// TwinCAT 3 PLC project AIR_Kinematics
// ProgramVersion: 3.1.4023.0
// libraries:
//   Standard, * (System)
//   Tc2_MC2, * (Beckhoff Automation GmbH)
//   Tc2_Standard, * (Beckhoff Automation GmbH)
//   Tc2_System, * (Beckhoff Automation GmbH)
//   Tc2_Utilities, * (Beckhoff Automation GmbH)
//   Tc3_Module, * (Beckhoff Automation GmbH)
// project tree:
//   DUTs/ ST_Trajectory.TcDUT
//   GVLs/ GVL.TcGVL
//   / PlcTask.TcTTO
//   POUs/ MAIN.TcPOU
//   StateData/ MoveState_t.TcDUT
// real-time tasks:
//   TASK PlcTask: cycle T#1ms, priority 1, ADS port 350
// motion (NC):
//   TASK NC-Task 1 SAF: cycle T#1ms, priority 4, ADS port 501
//   TASK NC-Task 1 SVB: cycle T#5ms, priority 8, ADS port 511
//   AXIS Axis 1 (id 1)
//     General: UnitName=Degree
//     Dynamic: AccelerationMaximum=1500, DecelerationMaximum=1500, Acceleration=2050.2, Deceleration=2050.2, Jerk=61506
//     Velo: RefSearch=2, RefSync=2, SlowManual=10, FastManual=50, Fast=136.68, Maximum=136.68
//     PositionAreaControl: Enable=false
//     TargetPosControl: Enable=false
//     OtherSettings: AllowMotionCmdToSlave=true
//     encoder EncType=19
//       EncPara: ScaleFactorNumerator=3.6, ScaleFactorDenominator=1048576, Offset=234, MaxCount=#xffffffff, ReferenceSystem=1
//         SoftEndMinControl: Enable=true, Range=-45
//         SoftEndMaxControl: Enable=true, Range=45
//     drive DrvType=16
//       DrvPara: MaxCount=#xffffffff, DriveControlDWord=#x00020000
//         Analog: VeloReferenz=150.348, VeloScale=32, TorqueSetpointScale=10, ScaleFactorActTorque=0.1
//         TimeComp: TaskDelayCycles=1
//     controller CtrType=1
//       CtrPara: PriorControlFactor=1
//         PosDiffControl: Enable=false
//         Observer: BandWidth=20
//   AXIS Axis 2 (id 2)
//     General: UnitName=Degree
//     Dynamic: AccelerationMaximum=1500, DecelerationMaximum=1500, Acceleration=2050.2, Deceleration=2050.2, Jerk=61506
//     Velo: RefSearch=2, RefSync=2, SlowManual=5, FastManual=50, Fast=136.68, Maximum=136.68
//     PositionAreaControl: Enable=false
//     TargetPosControl: Enable=false
//     OtherSettings: AllowMotionCmdToSlave=true
//     encoder EncType=19
//       EncPara: ScaleFactorNumerator=3.6, ScaleFactorDenominator=1048576, Offset=356.451663208008, Inverse=true, MaxCount=#xffffffff, ReferenceSystem=1
//         SoftEndMinControl: Enable=true, Range=-1
//         SoftEndMaxControl: Enable=true, Range=90
//     drive DrvType=16
//       DrvPara: Inverse=true, MaxCount=#xffffffff, DriveControlDWord=#x00020000
//         Analog: VeloReferenz=150.348, VeloScale=32, TorqueSetpointScale=10, ScaleFactorActTorque=0.1
//         TimeComp: TaskDelayCycles=1
//     controller CtrType=1
//       CtrPara: PriorControlFactor=1
//         PosDiffControl: Enable=false
//         Observer: BandWidth=20
//   AXIS Axis 3 (id 3)
//     General: UnitName=Degree
//     Dynamic: AccelerationMaximum=3000, DecelerationMaximum=3000, Acceleration=4369.5, Deceleration=4369.5, Jerk=131085
//     Velo: RefSearch=2, RefSync=2, SlowManual=20, FastManual=50, Fast=291.3, Maximum=291.3
//     PositionAreaControl: Enable=false
//     TargetPosControl: Enable=false
//     OtherSettings: AllowMotionCmdToSlave=true
//     encoder EncType=19
//       EncPara: ScaleFactorNumerator=3.6, ScaleFactorDenominator=1048576, Offset=-169.531800842285, MaxCount=#xffffffff, ReferenceSystem=1
//         SoftEndMinControl: Enable=true, Range=-90
//         SoftEndMaxControl: Enable=true, Range=90
//     drive DrvType=16
//       DrvPara: MaxCount=#xffffffff, DriveControlDWord=#x00020000
//         Analog: VeloReferenz=320.43, VeloScale=32, TorqueSetpointScale=10, ScaleFactorActTorque=0.1
//         TimeComp: TaskDelayCycles=1
//     controller CtrType=1
//       CtrPara: PriorControlFactor=1
//         PosDiffControl: Enable=false
//         Observer: BandWidth=20
//   AXIS elbow (id 4)
//     Dynamic: AccelerationMaximum=300, DecelerationMaximum=300, Acceleration=1793.71, Deceleration=1793.71, Jerk=271037
//     Velo: RefSearch=2, RefSync=2, SlowManual=5, FastManual=10, Maximum=100
//     PositionAreaControl: Enable=false
//     TargetPosControl: Enable=false
//     OtherSettings: AllowMotionCmdToSlave=true
//     encoder EncType=19
//       EncPara: ScaleFactorNumerator=19.073486328125, ScaleFactorDenominator=1000000, Offset=-205.2, MaxCount=#xffffffff, ReferenceSystem=1
//         SoftEndMinControl: Enable=true, Range=12.5
//         SoftEndMaxControl: Enable=true, Range=75
//     drive DrvType=16
//       DrvPara: MaxCount=#xffffffff
//         Analog: VeloReferenz=100, TorqueSetpointScale=10, ScaleFactorActTorque=0.1
//         TimeComp: TaskDelayCycles=1
//     controller CtrType=1
//       CtrPara: PriorControlFactor=1
//         PosDiffControl: Enable=false
//         Observer: BandWidth=20
//   AXIS roll (id 7)
//     Dynamic: AccelerationMaximum=30, DecelerationMaximum=30, Acceleration=75.75, Deceleration=75.75, Jerk=76507.5
//     Velo: RefSearch=1.5, RefSync=1.5, SlowManual=3.5, FastManual=7.5, Maximum=7.5
//     OtherSettings: AllowMotionCmdToSlave=true
//     encoder EncType=19
//       EncPara: ScaleFactorNumerator=2.846789, ScaleFactorDenominator=1000000, Offset=-11.48, MaxCount=#xffffffff, ReferenceSystem=1
//         SoftEndMinControl: Enable=true, Range=-15
//         SoftEndMaxControl: Enable=true, Range=15
//     drive DrvType=16
//       DrvPara: MaxCount=#xffffffff
//         Analog: VeloReferenz=7.5, TorqueSetpointScale=10, ScaleFactorActTorque=0.1
//         TimeComp: TaskDelayCycles=1
//     controller CtrType=1
//       CtrPara: PriorControlFactor=1
//         Observer: BandWidth=20
//   AXIS pitch (id 6)
//     Dynamic: AccelerationMaximum=30, DecelerationMaximum=30, Acceleration=75.75, Deceleration=75.75, Jerk=76507.5
//     Velo: RefSearch=1.5, RefSync=1.5, SlowManual=3.5, FastManual=7.5, Maximum=7.5
//     OtherSettings: AllowMotionCmdToSlave=true
//     encoder EncType=19
//       EncPara: ScaleFactorNumerator=2.846789, ScaleFactorDenominator=1000000, Offset=35, MaxCount=#xffffffff, ReferenceSystem=1
//         SoftEndMinControl: Enable=true, Range=-30
//         SoftEndMaxControl: Enable=true, Range=15
//     drive DrvType=16
//       DrvPara: MaxCount=#xffffffff
//         Analog: VeloReferenz=7.5, TorqueSetpointScale=10, ScaleFactorActTorque=0.1
//         TimeComp: TaskDelayCycles=1
//     controller CtrType=1
//       CtrPara: PriorControlFactor=1
//         Observer: BandWidth=20
//   AXIS yaw (id 5)
//     General: UnitName=Degree
//     Dynamic: AccelerationMaximum=5500, DecelerationMaximum=5500, Acceleration=2300, Deceleration=2300, Jerk=529000
//     Velo: Maximum=220
//     PositionAreaControl: Enable=false
//     OtherSettings: AllowMotionCmdToSlave=true
//     encoder EncType=19
//       EncPara: ScaleFactorNumerator=556.2698, ScaleFactorDenominator=1000000, MaxCount=#xffffffff
//         SoftEndMaxControl: Range=180
//     drive DrvType=16
//       DrvPara: MaxCount=#xffffffff
//         Analog: VeloReferenz=220, TorqueSetpointScale=10, ScaleFactorActTorque=0.1
//         TimeComp: TaskDelayCycles=1
//     controller CtrType=1
//       CtrPara: PriorControlFactor=1
//         PosDiffControl: Enable=false
//         Observer: BandWidth=20
// I/O:
//   DEVICE Device 5 (EtherCAT), AmsNetId 192.168.225.1.6.1
//     Term 12 (EK1100) [EK1100 EtherCAT Coupler (2A E-Bus)]
//       Term 13 (EL7211-0010) [EL7211-0010 1Ch. MDP742 Servo motor output stage with OCT (50V, 4.5A RMS)]
//       Term 14 (EL7211-0010) [EL7211-0010 1Ch. MDP742 Servo motor output stage with OCT (50V, 4.5A RMS)]
//       Term 15 (EL7211-0010) [EL7211-0010 1Ch. MDP742 Servo motor output stage with OCT (50V, 4.5A RMS)]
//       Term 16 (EL7211-0010) [EL7211-0010 1Ch. MDP742 Servo motor output stage with OCT (50V, 4.5A RMS)]
//       Term 17 (EL1008) [EL1008 8Ch. Dig. Input 24V, 3ms]
//       Term 18 (EL2008) [EL2008 8Ch. Dig. Output 24V, 0.5A]
//       Term 23 (EL9011) [EL9011 End Terminal]
//     Drive 19 (Capitan Drv) [Capitan Drv]
//     Drive 20 (Capitan Drv) [Capitan Drv]
//     Drive 21 (Capitan Drv) [Capitan Drv]
//     Drive 22 (Capitan Drv) [Capitan Drv]
// variable links:
//   NC-Task 1 SAF/Axes/Axis 1 <-> Device 5 (EtherCAT)/Term 12 (EK1100)/Term 13 (EL7211-0010)
//     Drive/Inputs/In/nDcOutputTime <-> InfoData/DcOutputShift
//     Drive/Inputs/In/nState1 <-> DRV Statusword/Statusword
//     Drive/Inputs/In/nState2 <-> DRV Statusword/Statusword @bit 8
//     Drive/Inputs/In/nState4 @bit 1 <-> WcState/InputToggle
//     Drive/Inputs/In/nState4 <-> WcState/WcState
//     Drive/Outputs/Out/nCtrl1 <-> DRV Controlword/Controlword
//     Drive/Outputs/Out/nCtrl2 <-> DRV Controlword/Controlword @bit 8
//     Drive/Outputs/Out/nDataOut2 <-> DRV Target velocity/Target velocity
//     Enc/Inputs/In/nDataIn1 <-> FB Position/Position
//     Enc/Inputs/In/nDcInputTime <-> InfoData/DcInputShift
//     Enc/Inputs/In/nState4 @bit 1 <-> WcState/InputToggle
//     Enc/Inputs/In/nState4 <-> WcState/WcState
//   NC-Task 1 SAF/Axes/Axis 2 <-> Device 5 (EtherCAT)/Term 12 (EK1100)/Term 14 (EL7211-0010)
//     Drive/Inputs/In/nDcOutputTime <-> InfoData/DcOutputShift
//     Drive/Inputs/In/nState1 <-> DRV Statusword/Statusword
//     Drive/Inputs/In/nState2 <-> DRV Statusword/Statusword @bit 8
//     Drive/Inputs/In/nState4 @bit 1 <-> WcState/InputToggle
//     Drive/Inputs/In/nState4 <-> WcState/WcState
//     Drive/Outputs/Out/nCtrl1 <-> DRV Controlword/Controlword
//     Drive/Outputs/Out/nCtrl2 <-> DRV Controlword/Controlword @bit 8
//     Drive/Outputs/Out/nDataOut2 <-> DRV Target velocity/Target velocity
//     Enc/Inputs/In/nDataIn1 <-> FB Position/Position
//     Enc/Inputs/In/nDcInputTime <-> InfoData/DcInputShift
//     Enc/Inputs/In/nState4 @bit 1 <-> WcState/InputToggle
//     Enc/Inputs/In/nState4 <-> WcState/WcState
//   NC-Task 1 SAF/Axes/Axis 3 <-> Device 5 (EtherCAT)/Term 12 (EK1100)/Term 16 (EL7211-0010)
//     Drive/Inputs/In/nDcOutputTime <-> InfoData/DcOutputShift
//     Drive/Inputs/In/nState1 <-> DRV Statusword/Statusword
//     Drive/Inputs/In/nState2 <-> DRV Statusword/Statusword @bit 8
//     Drive/Inputs/In/nState4 @bit 1 <-> WcState/InputToggle
//     Drive/Inputs/In/nState4 <-> WcState/WcState
//     Drive/Outputs/Out/nCtrl1 <-> DRV Controlword/Controlword
//     Drive/Outputs/Out/nCtrl2 <-> DRV Controlword/Controlword @bit 8
//     Drive/Outputs/Out/nDataOut2 <-> DRV Target velocity/Target velocity
//     Enc/Inputs/In/nDataIn1 <-> FB Position/Position
//     Enc/Inputs/In/nDcInputTime <-> InfoData/DcInputShift
//     Enc/Inputs/In/nState4 @bit 1 <-> WcState/InputToggle
//     Enc/Inputs/In/nState4 <-> WcState/WcState
//   NC-Task 1 SAF/Axes/elbow <-> Device 5 (EtherCAT)/Drive 19 (Capitan Drv)
//     Drive/Inputs/In/nState1 <-> TPDO 1 mapping parameter/Status Word
//     Drive/Inputs/In/nState2 <-> TPDO 1 mapping parameter/Status Word @bit 8
//     Drive/Inputs/In/nState4 @bit 1 <-> WcState/InputToggle
//     Drive/Inputs/In/nState4 <-> WcState/WcState
//     Drive/Inputs/In/nState5 <-> TPDO 1 mapping parameter/Operation mode display
//     Drive/Outputs/Out/nCtrl1 <-> RPDO 1 mapping parameter/Control Word
//     Drive/Outputs/Out/nCtrl2 <-> RPDO 1 mapping parameter/Control Word @bit 8
//     Drive/Outputs/Out/nCtrl5 <-> RPDO 1 mapping parameter/Operation mode
//     Drive/Outputs/Out/nDataOut1 <-> RPDO 1 mapping parameter/Position set-point
//     Drive/Outputs/Out/nDataOut2 <-> RPDO 1 mapping parameter/Velocity set-point
//     Enc/Inputs/In/nDataIn1 <-> TPDO 1 mapping parameter/Actual position
//     Enc/Inputs/In/nDataIn7 <-> TPDO 1 mapping parameter/Actual velocity
//     Enc/Inputs/In/nState4 @bit 1 <-> WcState/InputToggle
//     Enc/Inputs/In/nState4 <-> WcState/WcState
//   NC-Task 1 SAF/Axes/pitch <-> Device 5 (EtherCAT)/Drive 21 (Capitan Drv)
//     Drive/Inputs/In/nState1 <-> TPDO 1 mapping parameter/Status Word
//     Drive/Inputs/In/nState2 <-> TPDO 1 mapping parameter/Status Word @bit 8
//     Drive/Inputs/In/nState4 @bit 1 <-> WcState/InputToggle
//     Drive/Inputs/In/nState4 <-> WcState/WcState
//     Drive/Inputs/In/nState5 <-> TPDO 1 mapping parameter/Operation mode display
//     Drive/Outputs/Out/nCtrl1 <-> RPDO 1 mapping parameter/Control Word
//     Drive/Outputs/Out/nCtrl2 <-> RPDO 1 mapping parameter/Control Word @bit 8
//     Drive/Outputs/Out/nCtrl5 <-> RPDO 1 mapping parameter/Operation mode
//     Drive/Outputs/Out/nDataOut1 <-> RPDO 1 mapping parameter/Position set-point
//     Drive/Outputs/Out/nDataOut2 <-> RPDO 1 mapping parameter/Velocity set-point
//     Enc/Inputs/In/nDataIn1 <-> TPDO 1 mapping parameter/Actual position
//     Enc/Inputs/In/nDataIn7 <-> TPDO 1 mapping parameter/Actual velocity
//     Enc/Inputs/In/nState4 @bit 1 <-> WcState/InputToggle
//     Enc/Inputs/In/nState4 <-> WcState/WcState
//   NC-Task 1 SAF/Axes/roll <-> Device 5 (EtherCAT)/Drive 22 (Capitan Drv)
//     Drive/Inputs/In/nState1 <-> TPDO 1 mapping parameter/Status Word
//     Drive/Inputs/In/nState2 <-> TPDO 1 mapping parameter/Status Word @bit 8
//     Drive/Inputs/In/nState4 @bit 1 <-> WcState/InputToggle
//     Drive/Inputs/In/nState4 <-> WcState/WcState
//     Drive/Inputs/In/nState5 <-> TPDO 1 mapping parameter/Operation mode display
//     Drive/Outputs/Out/nCtrl1 <-> RPDO 1 mapping parameter/Control Word
//     Drive/Outputs/Out/nCtrl2 <-> RPDO 1 mapping parameter/Control Word @bit 8
//     Drive/Outputs/Out/nCtrl5 <-> RPDO 1 mapping parameter/Operation mode
//     Drive/Outputs/Out/nDataOut1 <-> RPDO 1 mapping parameter/Position set-point
//     Drive/Outputs/Out/nDataOut2 <-> RPDO 1 mapping parameter/Velocity set-point
//     Enc/Inputs/In/nDataIn1 <-> TPDO 1 mapping parameter/Actual position
//     Enc/Inputs/In/nDataIn7 <-> TPDO 1 mapping parameter/Actual velocity
//     Enc/Inputs/In/nState4 @bit 1 <-> WcState/InputToggle
//     Enc/Inputs/In/nState4 <-> WcState/WcState
//   NC-Task 1 SAF/Axes/yaw <-> Device 5 (EtherCAT)/Drive 20 (Capitan Drv)
//     Drive/Inputs/In/nState1 <-> TPDO 1 mapping parameter/Status Word
//     Drive/Inputs/In/nState2 <-> TPDO 1 mapping parameter/Status Word @bit 8
//     Drive/Inputs/In/nState4 @bit 1 <-> WcState/InputToggle
//     Drive/Inputs/In/nState4 <-> WcState/WcState
//     Drive/Inputs/In/nState5 <-> TPDO 1 mapping parameter/Operation mode display
//     Drive/Outputs/Out/nCtrl1 <-> RPDO 1 mapping parameter/Control Word
//     Drive/Outputs/Out/nCtrl2 <-> RPDO 1 mapping parameter/Control Word @bit 8
//     Drive/Outputs/Out/nCtrl5 <-> RPDO 1 mapping parameter/Operation mode
//     Drive/Outputs/Out/nDataOut1 <-> RPDO 1 mapping parameter/Position set-point
//     Drive/Outputs/Out/nDataOut2 <-> RPDO 1 mapping parameter/Velocity set-point
//     Enc/Inputs/In/nDataIn1 <-> TPDO 1 mapping parameter/Actual position
//     Enc/Inputs/In/nDataIn7 <-> TPDO 1 mapping parameter/Actual velocity
//     Enc/Inputs/In/nState4 @bit 1 <-> WcState/InputToggle
//     Enc/Inputs/In/nState4 <-> WcState/WcState
//   AIR_Kinematics/AIR_Kinematics Instance <-> NC-Task 1 SAF/Axes/Axis 1
//     PlcTask Inputs/GVL.EksenArm[1].NcToPlc <-> Outputs/ToPlc
//     PlcTask Outputs/GVL.EksenArm[1].PlcToNc <-> Inputs/FromPlc
//   AIR_Kinematics/AIR_Kinematics Instance <-> NC-Task 1 SAF/Axes/Axis 2
//     PlcTask Inputs/GVL.EksenArm[2].NcToPlc <-> Outputs/ToPlc
//     PlcTask Outputs/GVL.EksenArm[2].PlcToNc <-> Inputs/FromPlc
//   AIR_Kinematics/AIR_Kinematics Instance <-> NC-Task 1 SAF/Axes/Axis 3
//     PlcTask Inputs/GVL.EksenArm[3].NcToPlc <-> Outputs/ToPlc
//     PlcTask Outputs/GVL.EksenArm[3].PlcToNc <-> Inputs/FromPlc
//   AIR_Kinematics/AIR_Kinematics Instance <-> NC-Task 1 SAF/Axes/elbow
//     PlcTask Inputs/GVL.EksenArm[4].NcToPlc <-> Outputs/ToPlc
//     PlcTask Outputs/GVL.EksenArm[4].PlcToNc <-> Inputs/FromPlc
//   AIR_Kinematics/AIR_Kinematics Instance <-> NC-Task 1 SAF/Axes/pitch
//     PlcTask Inputs/GVL.EksenArm[6].NcToPlc <-> Outputs/ToPlc
//     PlcTask Outputs/GVL.EksenArm[6].PlcToNc <-> Inputs/FromPlc
//   AIR_Kinematics/AIR_Kinematics Instance <-> NC-Task 1 SAF/Axes/roll
//     PlcTask Inputs/GVL.EksenArm[5].NcToPlc <-> Outputs/ToPlc
//     PlcTask Outputs/GVL.EksenArm[5].PlcToNc <-> Inputs/FromPlc
//   AIR_Kinematics/AIR_Kinematics Instance <-> NC-Task 1 SAF/Axes/yaw
//     PlcTask Inputs/GVL.EksenArm[7].NcToPlc <-> Outputs/ToPlc
//     PlcTask Outputs/GVL.EksenArm[7].PlcToNc <-> Inputs/FromPlc

CONFIGURATION AIR_Kinematics
    RESOURCE PLC ON TwinCAT3
        TASK PlcTask(INTERVAL := T#1ms, PRIORITY := 1);
        PROGRAM MAIN WITH PlcTask : MAIN;
    END_RESOURCE
END_CONFIGURATION

// ---- DUTs/ST_Trajectory.TcDUT
TYPE ST_Trajectory :
STRUCT
	fPosition: LREAL;
	fVelocity: LREAL;
	fAcceleration: LREAL;
END_STRUCT
END_TYPE

// ---- StateData/MoveState_t.TcDUT
TYPE MoveState_t :
(
	MOVESTATE_INIT,
	MOVESTATE_ENABLE,
	MOVESTATE_FORWARD,
	MOVESTATE_BACKWARDS,
	MOVESTATE_BACKWARDSSLOW,
	MOVESTATE_NEWTARGETPOSITION,
	MOVESTATE_ERROR,
	MOVESTATE_RESET
);
END_TYPE

// ---- GVLs/GVL.TcGVL
VAR_GLOBAL CONSTANT
END_VAR

VAR_GLOBAL CONSTANT
	cnMaxAxis: INT := 7;
	cnMaxArrayLength: INT := 1500;
	Max_Row: INT := 3000;
END_VAR

VAR_GLOBAL

	PowerAxisArm	: ARRAY[1..7] OF TC2_MC2.MC_Power;
	MC_Move_1_Velocity: ARRAY[1..7] OF MC_MoveVelocity;
	MC_Move_2_Velocity: ARRAY[1..7] OF MC_MoveVelocity;
	EksenArm	: ARRAY[1..7] OF AXIS_REF;

	fGoalPos_Arm : ARRAY[1..7] OF LREAL ;
	fGoalVel_Arm : ARRAY[1..7] OF LREAL := [7(0)];
	fGoalAcc_Arm : ARRAY[1..7] OF LREAL := [7(0)];
	fActPose_Arm : ARRAY[1..7] OF LREAL ;
	fActVel_Arm: ARRAY[1..7] OF LREAL;
	
	bArmEnable: ARRAY [1..7] OF BOOL  := [7(TRUE)];
	bArmNegative: ARRAY[1..7] OF BOOL := [7(TRUE)];
	bArmPositive: ARRAY[1..7] OF BOOL := [7(TRUE)];
	
	SAVE_DATA: BOOL := FALSE;
	csvActPos: ARRAY[1..1500, 1..7] OF LREAL;
	csvActVel: ARRAY[1..1500, 1..7] OF LREAL;
	csvGoalPos: ARRAY[1..1500, 1..7] OF LREAL;
	csvGoalVel: ARRAY[1..1500, 1..7] OF LREAL;
	
	fArmOverride: REAL := 100;	
	
	bMove_1_Arm:  BOOL := FALSE;
	bMove_2_Arm:  BOOL := FALSE;
	
	Error_latch: ARRAY[1..7] OF UDINT ;
	
	axis_done_state: UDINT := 0;
	state_DONE: BOOL := FALSE;
	state_HALT: BOOL := FALSE;
	state_TIMEOUT: BOOL := FALSE;

	MC_Halt_1: MC_Halt;
	MC_Halt_2: MC_Halt;
	MC_Halt_3: MC_Halt;
	MC_Halt_4: MC_Halt;
	MC_Halt_5: MC_Halt;
	MC_Halt_6: MC_Halt;
	MC_Halt_7: MC_Halt;
	
	f_Halt_Dec_Arm : ARRAY[1..7] OF LREAL;
	fHalt_jerk: LREAL := 20;	
	
	fLastTimeStamp: UDINT;
	fActTimeStamp: UDINT;
	max_time_out: UDINT :=2000;
	
	nWriteArrayCount: INT := Max_Row;
	RefPos: ARRAY[1..Max_Row, 1..cnMaxAxis] OF LREAL;
	RefVel: ARRAY[1..Max_Row, 1..cnMaxAxis] OF LREAL;
	ActPos: ARRAY[1..Max_Row, 1..cnMaxAxis] OF LREAL;
	ActVel: ARRAY[1..Max_Row, 1..cnMaxAxis] OF LREAL;
	RefTrk: ARRAY[1..Max_Row, 1..cnMaxAxis] OF LREAL;
	ActTrk: ARRAY[1..Max_Row, 1..cnMaxAxis] OF LREAL;
	RefDrv: ARRAY[1..Max_Row, 1..cnMaxAxis] OF LREAL;
	ActDrv: ARRAY[1..Max_Row, 1..cnMaxAxis] OF LREAL;
	RefAcc: ARRAY[1..Max_Row, 1..cnMaxAxis] OF LREAL;
	ActAcc: ARRAY[1..Max_Row, 1..cnMaxAxis] OF LREAL;
	
	bLimitSwitch AT%I*: BOOL := FALSE;
	state_INIT : BOOL := TRUE;
	state_Eksen2_INIT : BOOL := TRUE;
END_VAR

// ---- POUs/MAIN.TcPOU
PROGRAM MAIN
VAR
	i: INT;
	error_counter: INT := 0;
	time_out_counter: UDINT :=0;
	num_of_axis: INT := 7;
	axis_index: INT := 0;
	online_counter: UDINT := 0;
	write_counter: UDINT := 1;
	
	fVel_Arm : ARRAY[1..7] OF LREAL := [7(0)];
	fAcc_Arm : ARRAY[1..7] OF LREAL := [7(0)];
	fDec_Arm : ARRAY[1..7] OF LREAL := [7(0)];
	fJerk_Arm : ARRAY[1..7] OF LREAL := [7(0)];
	fPos_Yaw : LREAL ;
	fDir_Arm : ARRAY[1..7] OF MC_DIRECTION;
	
	MC_Move_1_Absolute: ARRAY[1..7] OF MC_MoveAbsolute;
	MC_Move_2_Absolute: ARRAY[1..7] OF MC_MoveAbsolute;
	bMove_1_Arm_Abs: BOOL := FALSE;
	bMove_2_Arm_Abs: BOOL := FALSE;
	
	nState: INT := 930;
	bSetPos_Yaw: BOOL;
	MC_SetPosition_Yaw: MC_SetPosition;
END_VAR

ACT_Power();
//Mov_Absolute();

//IF state_INIT THEN
//	ACT_LimitSwitch();
//ELSE
	
IF fLastTimeStamp <> 0 AND (fActTimeStamp - fLastTimeStamp) = 0 THEN
	time_out_counter := time_out_counter + 1;
ELSE
	time_out_counter := 0;
END_IF

IF time_out_counter > max_time_out THEN
	state_TIMEOUT := TRUE;
	state_HALT := TRUE;
	fLastTimeStamp:= 0;
	fActTimeStamp:= 0;
	time_out_counter := 0;
	FOR axis_index:=1 TO num_of_axis DO
		f_Halt_Dec_Arm[axis_index] := EksenArm[axis_index].NcToPlc.ActAcc * 5;
		fVel_Arm[axis_index] := 0.0;
		fAcc_Arm[axis_index] := 0.0;
		fDec_Arm[axis_index] := 0.0;
	END_FOR
ELSE
	//////////////// SET DIRECTION \\\\\\\\\\\\\\\\\\\\\\

	FOR axis_index:=1 TO num_of_axis DO
		IF fGoalVel_Arm[axis_index] < 0 THEN
			fDir_Arm[axis_index] := MC_Negative_Direction;
		ELSE
			fDir_Arm[axis_index] := MC_Positive_Direction;
		END_IF
	END_FOR
	
	//////////////// SET PARAMETERS \\\\\\\\\\\\\\\\\\\\\\
	
	FOR axis_index:=1 TO num_of_axis DO	
		fVel_Arm[axis_index] := ABS(fGoalVel_Arm[axis_index]);
		fAcc_Arm[axis_index] := ABS(fGoalAcc_Arm[axis_index]);
		fDec_Arm[axis_index] := ABS(fGoalAcc_Arm[axis_index]);
	END_FOR	
END_IF

//////////////// FILL UP JOINT STATES \\\\\\\\\\\\\\\\\\\\\\

FOR axis_index:=1 TO num_of_axis DO	
	fActPose_Arm[axis_index] := EksenArm[axis_index].NcToPlc.ActPos;
	fActVel_Arm[axis_index] := EksenArm[axis_index].NcToPlc.ActVelo;
END_FOR	

//////////////// SAVE DATA \\\\\\\\\\\\\\\\\\\\\\

IF SAVE_DATA THEN
	IF (online_counter MOD 25) = 0 THEN
		FOR i:=1 TO 7 DO
			csvActPos[write_counter, i] := EksenArm[i].NcToPlc.ActPos;
			csvActVel[write_counter, i] := EksenArm[i].NcToPlc.ActVelo;
			csvGoalPos[write_counter, i] := fGoalPos_Arm[i];
			csvGoalVel[write_counter, i] := fGoalVel_Arm[i];
		END_FOR
		write_counter:= write_counter + 1;
	END_IF
	online_counter:= online_counter + 1;	
END_IF

////////////// CHECK ERROR STATE \\\\\\\\\\\\\\\\\\\\\\

//FOR error_counter:=1 TO num_of_axis DO
//	IF PowerAxisArm[error_counter].ErrorID <> 0 THEN
//		Error_latch[error_counter] := 100;
//		bMove_1_Arm := FALSE;
//		bMove_2_Arm := FALSE;
//		bRunBlocks := FALSE;
//		state_HALT := TRUE;
//		FOR halt_counter:=1 TO num_of_axis DO
//			f_Halt_Dec_Arm[halt_counter] := EksenArm[halt_counter].NcToPlc.ActAcc * 5;
//		END_FOR
//	END_IF
//END_FOR


////////////// SWITCH MOTION BLOCKS \\\\\\\\\\\\\\\\\\\\\\

IF bMove_1_Arm THEN
	bMove_1_Arm := FALSE;
	bMove_2_Arm := TRUE;
ELSE
	bMove_1_Arm := TRUE;
	bMove_2_Arm := FALSE;
END_IF


fLastTimeStamp := fActTimeStamp;

//END_IF

ACTION ACT_LimitSwitch:
IF EksenArm[2].NcToPlc.ActPos < 20.0 THEN
	Main.fVel_Arm[2] := 5.0;
	Main.fDir_Arm[2] := MC_Positive_Direction;
ELSE
	fVel_Arm[2] := 0.0;

	IF NOT bLimitSwitch THEN	
		fVel_Arm[7] := 20.0;
		Main.fDir_Arm[7] := MC_Negative_Direction;
	ELSE
		Main.bSetPos_Yaw := TRUE;	
		fVel_Arm[7] := 0.0;
		Mc_SetPosition_Yaw.Position := -120.0;
		state_INIT := FALSE;
	END_IF
END_IF

IF bMove_1_Arm THEN
	bMove_1_Arm := FALSE;
	bMove_2_Arm := TRUE;
ELSE
	bMove_1_Arm := TRUE;
	bMove_2_Arm := FALSE;
END_IF
END_ACTION

ACTION ACT_Power:
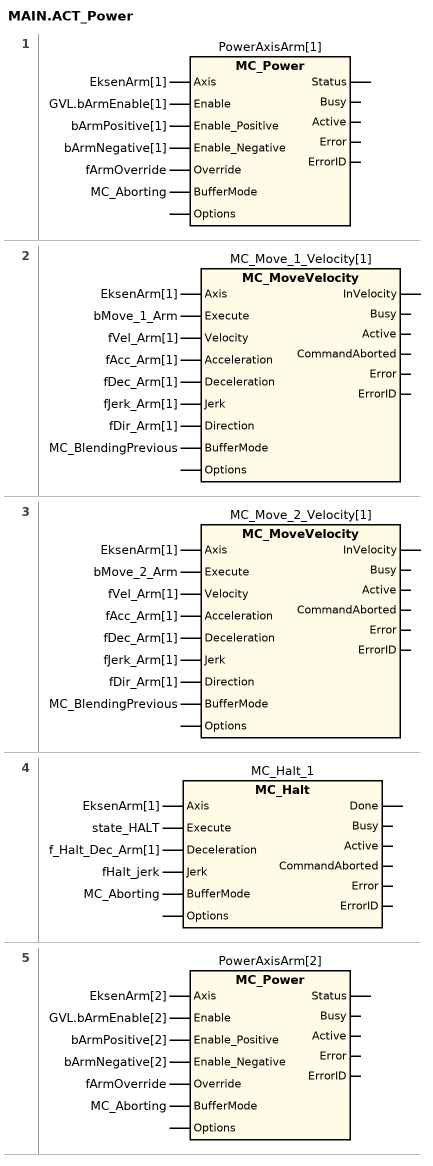
// NETWORK 1
PowerAxisArm[1](
    Axis := EksenArm[1],
    Enable := GVL.bArmEnable[1],
    Enable_Positive := bArmPositive[1],
    Enable_Negative := bArmNegative[1],
    Override := fArmOverride,
    BufferMode := MC_Aborting); // MC_Power

// NETWORK 2
MC_Move_1_Velocity[1](
    Axis := EksenArm[1],
    Execute := bMove_1_Arm,
    Velocity := fVel_Arm[1],
    Acceleration := fAcc_Arm[1],
    Deceleration := fDec_Arm[1],
    Jerk := fJerk_Arm[1],
    Direction := fDir_Arm[1],
    BufferMode := MC_BlendingPrevious); // MC_MoveVelocity

// NETWORK 3
MC_Move_2_Velocity[1](
    Axis := EksenArm[1],
    Execute := bMove_2_Arm,
    Velocity := fVel_Arm[1],
    Acceleration := fAcc_Arm[1],
    Deceleration := fDec_Arm[1],
    Jerk := fJerk_Arm[1],
    Direction := fDir_Arm[1],
    BufferMode := MC_BlendingPrevious); // MC_MoveVelocity

// NETWORK 4
MC_Halt_1(
    Axis := EksenArm[1],
    Execute := state_HALT,
    Deceleration := f_Halt_Dec_Arm[1],
    Jerk := fHalt_jerk,
    BufferMode := MC_Aborting); // MC_Halt

// NETWORK 5
PowerAxisArm[2](
    Axis := EksenArm[2],
    Enable := GVL.bArmEnable[2],
    Enable_Positive := bArmPositive[2],
    Enable_Negative := bArmNegative[2],
    Override := fArmOverride,
    BufferMode := MC_Aborting); // MC_Power

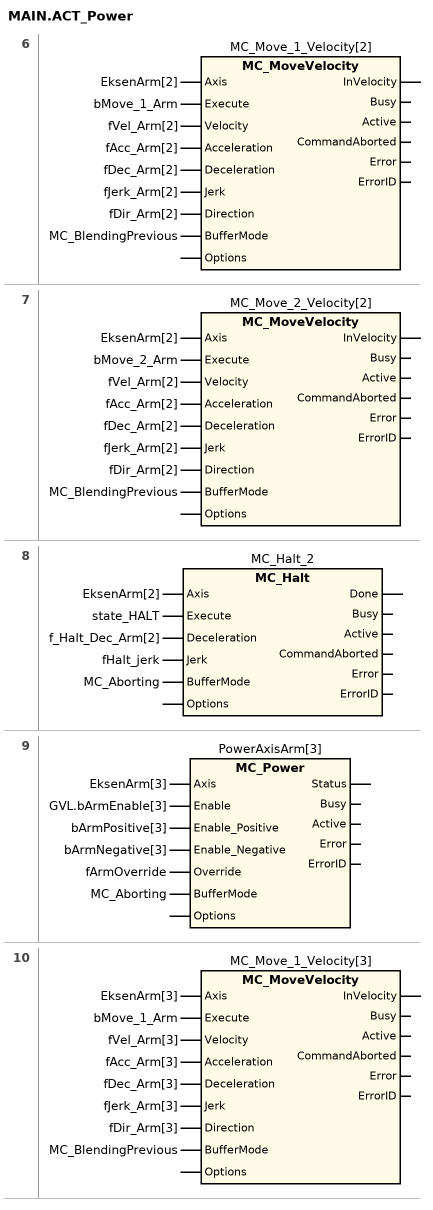
// NETWORK 6
MC_Move_1_Velocity[2](
    Axis := EksenArm[2],
    Execute := bMove_1_Arm,
    Velocity := fVel_Arm[2],
    Acceleration := fAcc_Arm[2],
    Deceleration := fDec_Arm[2],
    Jerk := fJerk_Arm[2],
    Direction := fDir_Arm[2],
    BufferMode := MC_BlendingPrevious); // MC_MoveVelocity

// NETWORK 7
MC_Move_2_Velocity[2](
    Axis := EksenArm[2],
    Execute := bMove_2_Arm,
    Velocity := fVel_Arm[2],
    Acceleration := fAcc_Arm[2],
    Deceleration := fDec_Arm[2],
    Jerk := fJerk_Arm[2],
    Direction := fDir_Arm[2],
    BufferMode := MC_BlendingPrevious); // MC_MoveVelocity

// NETWORK 8
MC_Halt_2(
    Axis := EksenArm[2],
    Execute := state_HALT,
    Deceleration := f_Halt_Dec_Arm[2],
    Jerk := fHalt_jerk,
    BufferMode := MC_Aborting); // MC_Halt

// NETWORK 9
PowerAxisArm[3](
    Axis := EksenArm[3],
    Enable := GVL.bArmEnable[3],
    Enable_Positive := bArmPositive[3],
    Enable_Negative := bArmNegative[3],
    Override := fArmOverride,
    BufferMode := MC_Aborting); // MC_Power

// NETWORK 10
MC_Move_1_Velocity[3](
    Axis := EksenArm[3],
    Execute := bMove_1_Arm,
    Velocity := fVel_Arm[3],
    Acceleration := fAcc_Arm[3],
    Deceleration := fDec_Arm[3],
    Jerk := fJerk_Arm[3],
    Direction := fDir_Arm[3],
    BufferMode := MC_BlendingPrevious); // MC_MoveVelocity

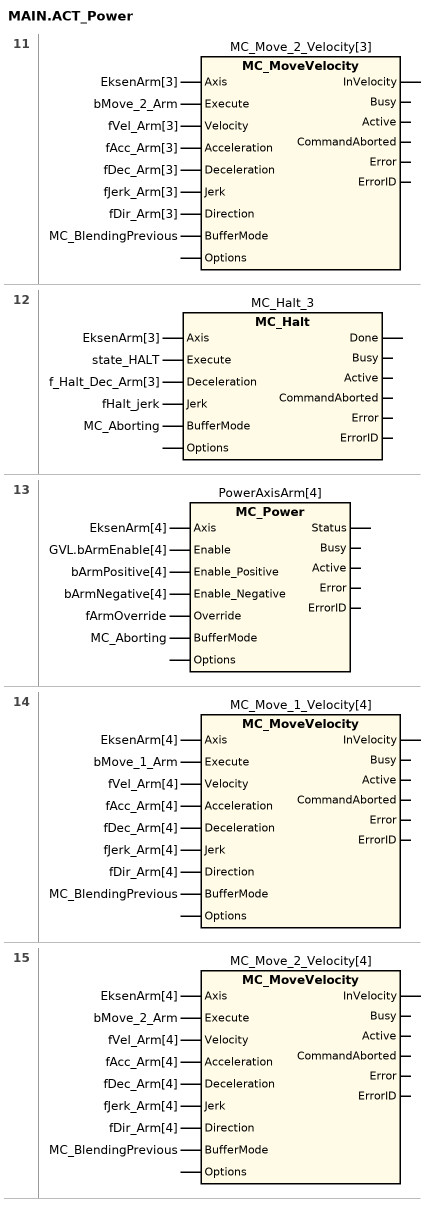
// NETWORK 11
MC_Move_2_Velocity[3](
    Axis := EksenArm[3],
    Execute := bMove_2_Arm,
    Velocity := fVel_Arm[3],
    Acceleration := fAcc_Arm[3],
    Deceleration := fDec_Arm[3],
    Jerk := fJerk_Arm[3],
    Direction := fDir_Arm[3],
    BufferMode := MC_BlendingPrevious); // MC_MoveVelocity

// NETWORK 12
MC_Halt_3(
    Axis := EksenArm[3],
    Execute := state_HALT,
    Deceleration := f_Halt_Dec_Arm[3],
    Jerk := fHalt_jerk,
    BufferMode := MC_Aborting); // MC_Halt

// NETWORK 13
PowerAxisArm[4](
    Axis := EksenArm[4],
    Enable := GVL.bArmEnable[4],
    Enable_Positive := bArmPositive[4],
    Enable_Negative := bArmNegative[4],
    Override := fArmOverride,
    BufferMode := MC_Aborting); // MC_Power

// NETWORK 14
MC_Move_1_Velocity[4](
    Axis := EksenArm[4],
    Execute := bMove_1_Arm,
    Velocity := fVel_Arm[4],
    Acceleration := fAcc_Arm[4],
    Deceleration := fDec_Arm[4],
    Jerk := fJerk_Arm[4],
    Direction := fDir_Arm[4],
    BufferMode := MC_BlendingPrevious); // MC_MoveVelocity

// NETWORK 15
MC_Move_2_Velocity[4](
    Axis := EksenArm[4],
    Execute := bMove_2_Arm,
    Velocity := fVel_Arm[4],
    Acceleration := fAcc_Arm[4],
    Deceleration := fDec_Arm[4],
    Jerk := fJerk_Arm[4],
    Direction := fDir_Arm[4],
    BufferMode := MC_BlendingPrevious); // MC_MoveVelocity

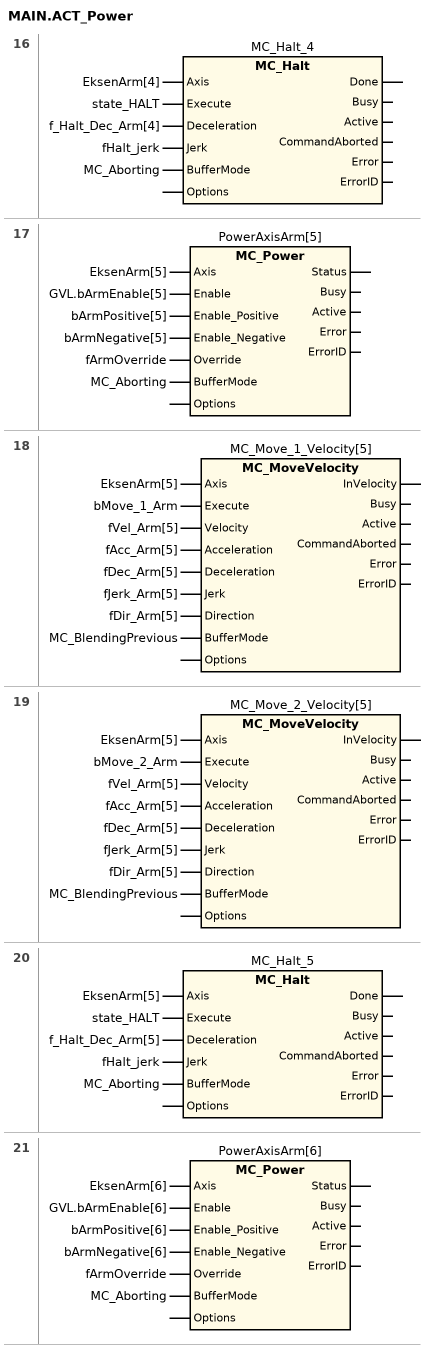
// NETWORK 16
MC_Halt_4(
    Axis := EksenArm[4],
    Execute := state_HALT,
    Deceleration := f_Halt_Dec_Arm[4],
    Jerk := fHalt_jerk,
    BufferMode := MC_Aborting); // MC_Halt

// NETWORK 17
PowerAxisArm[5](
    Axis := EksenArm[5],
    Enable := GVL.bArmEnable[5],
    Enable_Positive := bArmPositive[5],
    Enable_Negative := bArmNegative[5],
    Override := fArmOverride,
    BufferMode := MC_Aborting); // MC_Power

// NETWORK 18
MC_Move_1_Velocity[5](
    Axis := EksenArm[5],
    Execute := bMove_1_Arm,
    Velocity := fVel_Arm[5],
    Acceleration := fAcc_Arm[5],
    Deceleration := fDec_Arm[5],
    Jerk := fJerk_Arm[5],
    Direction := fDir_Arm[5],
    BufferMode := MC_BlendingPrevious); // MC_MoveVelocity

// NETWORK 19
MC_Move_2_Velocity[5](
    Axis := EksenArm[5],
    Execute := bMove_2_Arm,
    Velocity := fVel_Arm[5],
    Acceleration := fAcc_Arm[5],
    Deceleration := fDec_Arm[5],
    Jerk := fJerk_Arm[5],
    Direction := fDir_Arm[5],
    BufferMode := MC_BlendingPrevious); // MC_MoveVelocity

// NETWORK 20
MC_Halt_5(
    Axis := EksenArm[5],
    Execute := state_HALT,
    Deceleration := f_Halt_Dec_Arm[5],
    Jerk := fHalt_jerk,
    BufferMode := MC_Aborting); // MC_Halt

// NETWORK 21
PowerAxisArm[6](
    Axis := EksenArm[6],
    Enable := GVL.bArmEnable[6],
    Enable_Positive := bArmPositive[6],
    Enable_Negative := bArmNegative[6],
    Override := fArmOverride,
    BufferMode := MC_Aborting); // MC_Power

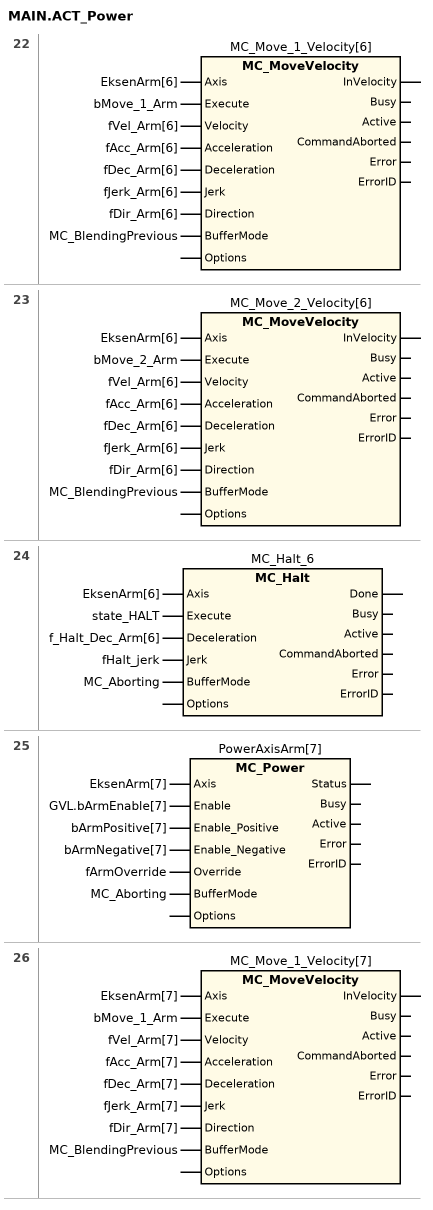
// NETWORK 22
MC_Move_1_Velocity[6](
    Axis := EksenArm[6],
    Execute := bMove_1_Arm,
    Velocity := fVel_Arm[6],
    Acceleration := fAcc_Arm[6],
    Deceleration := fDec_Arm[6],
    Jerk := fJerk_Arm[6],
    Direction := fDir_Arm[6],
    BufferMode := MC_BlendingPrevious); // MC_MoveVelocity

// NETWORK 23
MC_Move_2_Velocity[6](
    Axis := EksenArm[6],
    Execute := bMove_2_Arm,
    Velocity := fVel_Arm[6],
    Acceleration := fAcc_Arm[6],
    Deceleration := fDec_Arm[6],
    Jerk := fJerk_Arm[6],
    Direction := fDir_Arm[6],
    BufferMode := MC_BlendingPrevious); // MC_MoveVelocity

// NETWORK 24
MC_Halt_6(
    Axis := EksenArm[6],
    Execute := state_HALT,
    Deceleration := f_Halt_Dec_Arm[6],
    Jerk := fHalt_jerk,
    BufferMode := MC_Aborting); // MC_Halt

// NETWORK 25
PowerAxisArm[7](
    Axis := EksenArm[7],
    Enable := GVL.bArmEnable[7],
    Enable_Positive := bArmPositive[7],
    Enable_Negative := bArmNegative[7],
    Override := fArmOverride,
    BufferMode := MC_Aborting); // MC_Power

// NETWORK 26
MC_Move_1_Velocity[7](
    Axis := EksenArm[7],
    Execute := bMove_1_Arm,
    Velocity := fVel_Arm[7],
    Acceleration := fAcc_Arm[7],
    Deceleration := fDec_Arm[7],
    Jerk := fJerk_Arm[7],
    Direction := fDir_Arm[7],
    BufferMode := MC_BlendingPrevious); // MC_MoveVelocity

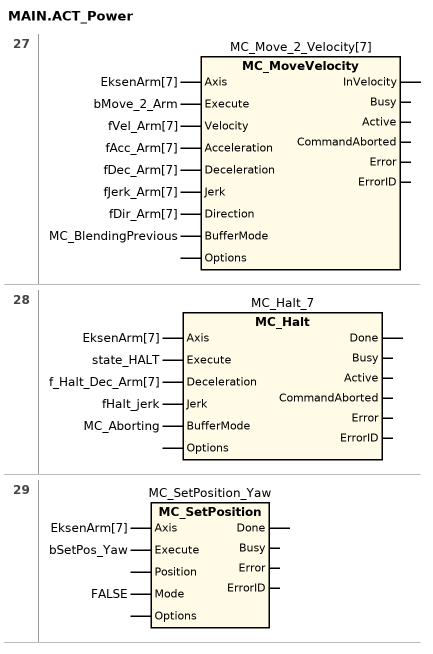
// NETWORK 27
MC_Move_2_Velocity[7](
    Axis := EksenArm[7],
    Execute := bMove_2_Arm,
    Velocity := fVel_Arm[7],
    Acceleration := fAcc_Arm[7],
    Deceleration := fDec_Arm[7],
    Jerk := fJerk_Arm[7],
    Direction := fDir_Arm[7],
    BufferMode := MC_BlendingPrevious); // MC_MoveVelocity

// NETWORK 28
MC_Halt_7(
    Axis := EksenArm[7],
    Execute := state_HALT,
    Deceleration := f_Halt_Dec_Arm[7],
    Jerk := fHalt_jerk,
    BufferMode := MC_Aborting); // MC_Halt

// NETWORK 29
MC_SetPosition_Yaw(Axis := EksenArm[7], Execute := bSetPos_Yaw, Mode := FALSE); // MC_SetPosition
END_ACTION

ACTION Mov_Absolute:
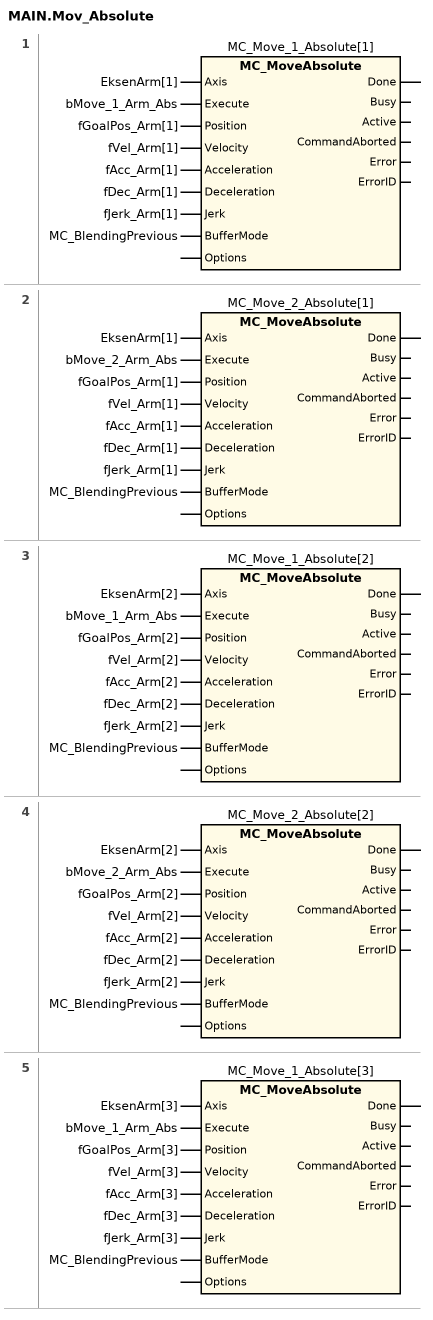
// NETWORK 1
MC_Move_1_Absolute[1](
    Axis := EksenArm[1],
    Execute := bMove_1_Arm_Abs,
    Position := fGoalPos_Arm[1],
    Velocity := fVel_Arm[1],
    Acceleration := fAcc_Arm[1],
    Deceleration := fDec_Arm[1],
    Jerk := fJerk_Arm[1],
    BufferMode := MC_BlendingPrevious); // MC_MoveAbsolute

// NETWORK 2
MC_Move_2_Absolute[1](
    Axis := EksenArm[1],
    Execute := bMove_2_Arm_Abs,
    Position := fGoalPos_Arm[1],
    Velocity := fVel_Arm[1],
    Acceleration := fAcc_Arm[1],
    Deceleration := fDec_Arm[1],
    Jerk := fJerk_Arm[1],
    BufferMode := MC_BlendingPrevious); // MC_MoveAbsolute

// NETWORK 3
MC_Move_1_Absolute[2](
    Axis := EksenArm[2],
    Execute := bMove_1_Arm_Abs,
    Position := fGoalPos_Arm[2],
    Velocity := fVel_Arm[2],
    Acceleration := fAcc_Arm[2],
    Deceleration := fDec_Arm[2],
    Jerk := fJerk_Arm[2],
    BufferMode := MC_BlendingPrevious); // MC_MoveAbsolute

// NETWORK 4
MC_Move_2_Absolute[2](
    Axis := EksenArm[2],
    Execute := bMove_2_Arm_Abs,
    Position := fGoalPos_Arm[2],
    Velocity := fVel_Arm[2],
    Acceleration := fAcc_Arm[2],
    Deceleration := fDec_Arm[2],
    Jerk := fJerk_Arm[2],
    BufferMode := MC_BlendingPrevious); // MC_MoveAbsolute

// NETWORK 5
MC_Move_1_Absolute[3](
    Axis := EksenArm[3],
    Execute := bMove_1_Arm_Abs,
    Position := fGoalPos_Arm[3],
    Velocity := fVel_Arm[3],
    Acceleration := fAcc_Arm[3],
    Deceleration := fDec_Arm[3],
    Jerk := fJerk_Arm[3],
    BufferMode := MC_BlendingPrevious); // MC_MoveAbsolute

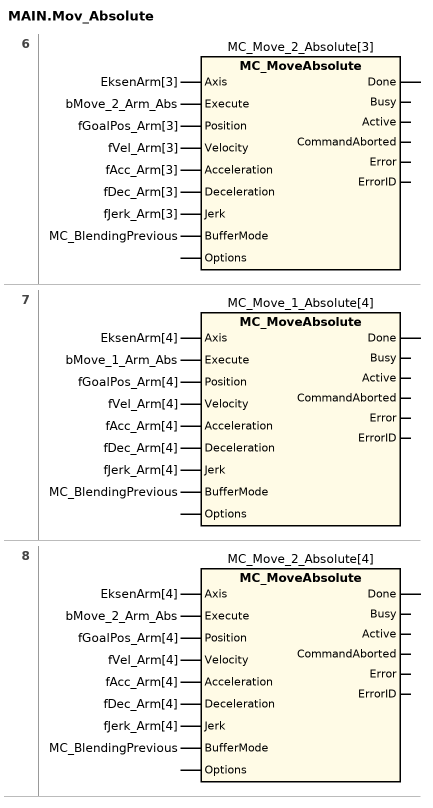
// NETWORK 6
MC_Move_2_Absolute[3](
    Axis := EksenArm[3],
    Execute := bMove_2_Arm_Abs,
    Position := fGoalPos_Arm[3],
    Velocity := fVel_Arm[3],
    Acceleration := fAcc_Arm[3],
    Deceleration := fDec_Arm[3],
    Jerk := fJerk_Arm[3],
    BufferMode := MC_BlendingPrevious); // MC_MoveAbsolute

// NETWORK 7
MC_Move_1_Absolute[4](
    Axis := EksenArm[4],
    Execute := bMove_1_Arm_Abs,
    Position := fGoalPos_Arm[4],
    Velocity := fVel_Arm[4],
    Acceleration := fAcc_Arm[4],
    Deceleration := fDec_Arm[4],
    Jerk := fJerk_Arm[4],
    BufferMode := MC_BlendingPrevious); // MC_MoveAbsolute

// NETWORK 8
MC_Move_2_Absolute[4](
    Axis := EksenArm[4],
    Execute := bMove_2_Arm_Abs,
    Position := fGoalPos_Arm[4],
    Velocity := fVel_Arm[4],
    Acceleration := fAcc_Arm[4],
    Deceleration := fDec_Arm[4],
    Jerk := fJerk_Arm[4],
    BufferMode := MC_BlendingPrevious); // MC_MoveAbsolute
END_ACTION

END_PROGRAM
